// TIA Portal V21 export
TYPE "coneCrusherHMI"
   STRUCT
      cmd : Struct
         cmdWord : Word;
      END_STRUCT;
      sta : Struct
         statusDWord : DWord;
         "step" : USInt;
         stepTime : LTime;
         almDWord { S7_SetPoint := 'True'} : DWord;
         stopCtx : "stopCtxHMI";
      END_STRUCT;
   END_STRUCT;
END_TYPE
